{attribute 'GeneratedUsingTerminal: EL6740-0010-0000'}
{attribute addProperty BoxType "EL6740-0010-0000"}
{attribute addProperty Id "EtcSlaveTerminalBaseStatusAT %I*Status_EF5E6C280InputsEMPTY_STRUCTURE0ControlAT %Q*Control_883019540OutputsEMPTY_STRUCTURE0WcStateAT %I*WcState_9091E0EB2InfoDataAT %I*InfoData_32EB74EA10"}
{attribute addProperty CRC "2629842823"}
{attribute addProperty Size "12"}
TYPE EL6740_9CC03787 EXTENDS EtcSlaveTerminalBase :
STRUCT
	{attribute addProperty Name "Status"}
	Status : Status_EF5E6C28;
	{attribute addProperty Name "Inputs"}
	Inputs : EMPTY_STRUCTURE;
	{attribute addProperty Name "Control"}
	Control : Control_88301954;
	{attribute addProperty Name "Outputs"}
	Outputs : EMPTY_STRUCTURE;
	{attribute addProperty Name "WcState"}
	WcState : WcState_9091E0EB;
	{attribute addProperty Name "InfoData"}
	InfoData : InfoData_32EB74EA;
END_STRUCT
END_TYPE

(* stored: Version 1.2.0.0, ProductVersion 3.1.4024.9
   DUT EL6740_9CC03787: Id {fc9fa39f-599f-4e31-852e-791303b65279} *)
